// TwinCAT 3 PLC project Plc
// ProgramVersion: 3.1.4023.0
// libraries:
//   Tc2_Standard, * (Beckhoff Automation GmbH)
//   Tc2_System, * (Beckhoff Automation GmbH)
//   Tc3_Module, * (Beckhoff Automation GmbH)
// project tree:
//   / PlcTask.TcTTO (not stored)
//   DUTs/IO/PdoEntries/ Status_3D84275F.TcDUT, Ctrl_1EFB4D3B.TcDUT
//   DUTs/IO/PDOs/ InfoData_6F19DB2B.TcDUT (not stored), COM_TxPDO_Map_Inputs_Channel_3801C95E.TcDUT, COM_TxPDO_Map_Inputs_Channel_6C2FC202.TcDUT, COM_RxPDO_Map_Outputs_Channel_EADA2E0D.TcDUT, COM_RxPDO_Map_Outputs_Channel_5D00B5E7.TcDUT, WcState_9091E0EB.TcDUT, InfoData_32EB74EA.TcDUT, InfoData_E68C61CD.TcDUT (not stored), WcState_0B2B16F9.TcDUT (not stored), InfoData_2A97D6CF.TcDUT (not stored), Inputs_A65FACA4.TcDUT (not stored), Outputs_23C0ED1D.TcDUT (not stored)
//   DUTs/IO/Boxes/ EK1100_1FC0878B.TcDUT (not stored), EL6002_642836E0.TcDUT
//   DUTs/IO/Devices/ SyncUnitTask_2D604ED5.TcDUT (not stored), SyncUnitTasks_6FEB8257.TcDUT (not stored), SyncUnits_99E584AF.TcDUT (not stored)
//   DUTs/IO/Topology/ Term_1_EK1100_40465B6B.TcDUT (not stored), Device_1_EtherCAT_B7DDB641.TcDUT (not stored)
//   DUTs/IO/Base/ EtcSlaveBase_82538BE2.TcDUT (not stored), EtcSlaveBase_82538BE2.TcDUT (not stored), EtcSlaveBase_82538BE2.TcDUT (not stored), EtcSlaveTerminalBase_947E5A46.TcDUT (not stored), EtcSlaveBoxBase_77A0E4A7.TcDUT (not stored), EtcSlaveEndTerminalBase_866C7F0C.TcDUT (not stored), InputBase_8311D824.TcDUT (not stored), OutputBase_10CEE7DE.TcDUT (not stored), EtcMasterBase_62654B43.TcDUT (not stored)
//   GVLs/ GVL_iXlinker.TcGVL (not stored)
// real-time tasks:
//   TASK PlcTask: cycle T#10ms, priority 20, ADS port 350
// I/O:
//   DEVICE Device 1 (EtherCAT), AmsNetId 172.20.30.238.2.1
//     Term 1 (EK1100) [EK1100 EtherCAT Coupler (2A E-Bus)]
//       Term 2 (EL6002) [EL6002 Interface 2Ch. (RS232)]
// variable links:
//   Plc/Plc Instance <-> Device 1 (EtherCAT)/Term 1 (EK1100)
//     PlcTask Inputs/GVL_iXlinker.Device_1_EtherCAT.Term_1_EK1100.InfoData.State <-> InfoData/State
//   Plc/Plc Instance <-> Device 1 (EtherCAT)/Term 1 (EK1100)/Term 2 (EL6002)
//     PlcTask Inputs/GVL_iXlinker.Device_1_EtherCAT.Term_1_EK1100.Term_2_EL6002.COM_TxPDO_Map_Inputs_Channel_1.Status/Transmit_accepted <-> COM TxPDO-Map Inputs Channel 1/Status/Transmit accepted
//     PlcTask Inputs/GVL_iXlinker.Device_1_EtherCAT.Term_1_EK1100.Term_2_EL6002.COM_TxPDO_Map_Inputs_Channel_1.Status/Receive_request <-> COM TxPDO-Map Inputs Channel 1/Status/Receive request
//     PlcTask Inputs/GVL_iXlinker.Device_1_EtherCAT.Term_1_EK1100.Term_2_EL6002.COM_TxPDO_Map_Inputs_Channel_1.Status/Init_accepted <-> COM TxPDO-Map Inputs Channel 1/Status/Init accepted
//     PlcTask Inputs/GVL_iXlinker.Device_1_EtherCAT.Term_1_EK1100.Term_2_EL6002.COM_TxPDO_Map_Inputs_Channel_1.Status/Buffer_full <-> COM TxPDO-Map Inputs Channel 1/Status/Buffer full
//     PlcTask Inputs/GVL_iXlinker.Device_1_EtherCAT.Term_1_EK1100.Term_2_EL6002.COM_TxPDO_Map_Inputs_Channel_1.Status/Parity_error <-> COM TxPDO-Map Inputs Channel 1/Status/Parity error
//     PlcTask Inputs/GVL_iXlinker.Device_1_EtherCAT.Term_1_EK1100.Term_2_EL6002.COM_TxPDO_Map_Inputs_Channel_1.Status/Framing_error <-> COM TxPDO-Map Inputs Channel 1/Status/Framing error
//     PlcTask Inputs/GVL_iXlinker.Device_1_EtherCAT.Term_1_EK1100.Term_2_EL6002.COM_TxPDO_Map_Inputs_Channel_1.Status/Overrun_error <-> COM TxPDO-Map Inputs Channel 1/Status/Overrun error
//     PlcTask Inputs/GVL_iXlinker.Device_1_EtherCAT.Term_1_EK1100.Term_2_EL6002.COM_TxPDO_Map_Inputs_Channel_1.Status/Input_length <-> COM TxPDO-Map Inputs Channel 1/Status/Input length
//     PlcTask Inputs/GVL_iXlinker.Device_1_EtherCAT.Term_1_EK1100.Term_2_EL6002.COM_TxPDO_Map_Inputs_Channel_1.Data_In[0] <-> COM TxPDO-Map Inputs Channel 1/Data In 0
//     PlcTask Inputs/GVL_iXlinker.Device_1_EtherCAT.Term_1_EK1100.Term_2_EL6002.COM_TxPDO_Map_Inputs_Channel_1.Data_In[1] <-> COM TxPDO-Map Inputs Channel 1/Data In 1
//     PlcTask Inputs/GVL_iXlinker.Device_1_EtherCAT.Term_1_EK1100.Term_2_EL6002.COM_TxPDO_Map_Inputs_Channel_1.Data_In[2] <-> COM TxPDO-Map Inputs Channel 1/Data In 2
//     PlcTask Inputs/GVL_iXlinker.Device_1_EtherCAT.Term_1_EK1100.Term_2_EL6002.COM_TxPDO_Map_Inputs_Channel_1.Data_In[3] <-> COM TxPDO-Map Inputs Channel 1/Data In 3
//     PlcTask Inputs/GVL_iXlinker.Device_1_EtherCAT.Term_1_EK1100.Term_2_EL6002.COM_TxPDO_Map_Inputs_Channel_1.Data_In[4] <-> COM TxPDO-Map Inputs Channel 1/Data In 4
//     PlcTask Inputs/GVL_iXlinker.Device_1_EtherCAT.Term_1_EK1100.Term_2_EL6002.COM_TxPDO_Map_Inputs_Channel_1.Data_In[5] <-> COM TxPDO-Map Inputs Channel 1/Data In 5
//     PlcTask Inputs/GVL_iXlinker.Device_1_EtherCAT.Term_1_EK1100.Term_2_EL6002.COM_TxPDO_Map_Inputs_Channel_1.Data_In[6] <-> COM TxPDO-Map Inputs Channel 1/Data In 6
//     PlcTask Inputs/GVL_iXlinker.Device_1_EtherCAT.Term_1_EK1100.Term_2_EL6002.COM_TxPDO_Map_Inputs_Channel_1.Data_In[7] <-> COM TxPDO-Map Inputs Channel 1/Data In 7
//     PlcTask Inputs/GVL_iXlinker.Device_1_EtherCAT.Term_1_EK1100.Term_2_EL6002.COM_TxPDO_Map_Inputs_Channel_1.Data_In[8] <-> COM TxPDO-Map Inputs Channel 1/Data In 8
//     PlcTask Inputs/GVL_iXlinker.Device_1_EtherCAT.Term_1_EK1100.Term_2_EL6002.COM_TxPDO_Map_Inputs_Channel_1.Data_In[9] <-> COM TxPDO-Map Inputs Channel 1/Data In 9
//     PlcTask Inputs/GVL_iXlinker.Device_1_EtherCAT.Term_1_EK1100.Term_2_EL6002.COM_TxPDO_Map_Inputs_Channel_1.Data_In[10] <-> COM TxPDO-Map Inputs Channel 1/Data In 10
//     PlcTask Inputs/GVL_iXlinker.Device_1_EtherCAT.Term_1_EK1100.Term_2_EL6002.COM_TxPDO_Map_Inputs_Channel_1.Data_In[11] <-> COM TxPDO-Map Inputs Channel 1/Data In 11
//     PlcTask Inputs/GVL_iXlinker.Device_1_EtherCAT.Term_1_EK1100.Term_2_EL6002.COM_TxPDO_Map_Inputs_Channel_1.Data_In[12] <-> COM TxPDO-Map Inputs Channel 1/Data In 12
//     PlcTask Inputs/GVL_iXlinker.Device_1_EtherCAT.Term_1_EK1100.Term_2_EL6002.COM_TxPDO_Map_Inputs_Channel_1.Data_In[13] <-> COM TxPDO-Map Inputs Channel 1/Data In 13
//     PlcTask Inputs/GVL_iXlinker.Device_1_EtherCAT.Term_1_EK1100.Term_2_EL6002.COM_TxPDO_Map_Inputs_Channel_1.Data_In[14] <-> COM TxPDO-Map Inputs Channel 1/Data In 14
//     PlcTask Inputs/GVL_iXlinker.Device_1_EtherCAT.Term_1_EK1100.Term_2_EL6002.COM_TxPDO_Map_Inputs_Channel_1.Data_In[15] <-> COM TxPDO-Map Inputs Channel 1/Data In 15
//     PlcTask Inputs/GVL_iXlinker.Device_1_EtherCAT.Term_1_EK1100.Term_2_EL6002.COM_TxPDO_Map_Inputs_Channel_1.Data_In[16] <-> COM TxPDO-Map Inputs Channel 1/Data In 16
//     PlcTask Inputs/GVL_iXlinker.Device_1_EtherCAT.Term_1_EK1100.Term_2_EL6002.COM_TxPDO_Map_Inputs_Channel_1.Data_In[17] <-> COM TxPDO-Map Inputs Channel 1/Data In 17
//     PlcTask Inputs/GVL_iXlinker.Device_1_EtherCAT.Term_1_EK1100.Term_2_EL6002.COM_TxPDO_Map_Inputs_Channel_1.Data_In[18] <-> COM TxPDO-Map Inputs Channel 1/Data In 18
//     PlcTask Inputs/GVL_iXlinker.Device_1_EtherCAT.Term_1_EK1100.Term_2_EL6002.COM_TxPDO_Map_Inputs_Channel_1.Data_In[19] <-> COM TxPDO-Map Inputs Channel 1/Data In 19
//     PlcTask Inputs/GVL_iXlinker.Device_1_EtherCAT.Term_1_EK1100.Term_2_EL6002.COM_TxPDO_Map_Inputs_Channel_1.Data_In[20] <-> COM TxPDO-Map Inputs Channel 1/Data In 20
//     PlcTask Inputs/GVL_iXlinker.Device_1_EtherCAT.Term_1_EK1100.Term_2_EL6002.COM_TxPDO_Map_Inputs_Channel_1.Data_In[21] <-> COM TxPDO-Map Inputs Channel 1/Data In 21
//     PlcTask Inputs/GVL_iXlinker.Device_1_EtherCAT.Term_1_EK1100.Term_2_EL6002.COM_TxPDO_Map_Inputs_Channel_2.Data_In[0] <-> COM TxPDO-Map Inputs Channel 2/Data In 0
//     PlcTask Inputs/GVL_iXlinker.Device_1_EtherCAT.Term_1_EK1100.Term_2_EL6002.COM_TxPDO_Map_Inputs_Channel_2.Data_In[1] <-> COM TxPDO-Map Inputs Channel 2/Data In 1
//     PlcTask Inputs/GVL_iXlinker.Device_1_EtherCAT.Term_1_EK1100.Term_2_EL6002.COM_TxPDO_Map_Inputs_Channel_2.Data_In[2] <-> COM TxPDO-Map Inputs Channel 2/Data In 2
//     PlcTask Inputs/GVL_iXlinker.Device_1_EtherCAT.Term_1_EK1100.Term_2_EL6002.COM_TxPDO_Map_Inputs_Channel_2.Data_In[3] <-> COM TxPDO-Map Inputs Channel 2/Data In 3
//     PlcTask Inputs/GVL_iXlinker.Device_1_EtherCAT.Term_1_EK1100.Term_2_EL6002.COM_TxPDO_Map_Inputs_Channel_2.Data_In[4] <-> COM TxPDO-Map Inputs Channel 2/Data In 4
//     PlcTask Inputs/GVL_iXlinker.Device_1_EtherCAT.Term_1_EK1100.Term_2_EL6002.COM_TxPDO_Map_Inputs_Channel_2.Data_In[5] <-> COM TxPDO-Map Inputs Channel 2/Data In 5
//     PlcTask Inputs/GVL_iXlinker.Device_1_EtherCAT.Term_1_EK1100.Term_2_EL6002.COM_TxPDO_Map_Inputs_Channel_2.Data_In[6] <-> COM TxPDO-Map Inputs Channel 2/Data In 6
//     PlcTask Inputs/GVL_iXlinker.Device_1_EtherCAT.Term_1_EK1100.Term_2_EL6002.COM_TxPDO_Map_Inputs_Channel_2.Data_In[7] <-> COM TxPDO-Map Inputs Channel 2/Data In 7
//     PlcTask Inputs/GVL_iXlinker.Device_1_EtherCAT.Term_1_EK1100.Term_2_EL6002.COM_TxPDO_Map_Inputs_Channel_2.Data_In[8] <-> COM TxPDO-Map Inputs Channel 2/Data In 8
//     PlcTask Inputs/GVL_iXlinker.Device_1_EtherCAT.Term_1_EK1100.Term_2_EL6002.COM_TxPDO_Map_Inputs_Channel_2.Data_In[9] <-> COM TxPDO-Map Inputs Channel 2/Data In 9
//     PlcTask Inputs/GVL_iXlinker.Device_1_EtherCAT.Term_1_EK1100.Term_2_EL6002.COM_TxPDO_Map_Inputs_Channel_2.Data_In[10] <-> COM TxPDO-Map Inputs Channel 2/Data In 10
//     PlcTask Inputs/GVL_iXlinker.Device_1_EtherCAT.Term_1_EK1100.Term_2_EL6002.COM_TxPDO_Map_Inputs_Channel_2.Data_In[11] <-> COM TxPDO-Map Inputs Channel 2/Data In 11
//     PlcTask Inputs/GVL_iXlinker.Device_1_EtherCAT.Term_1_EK1100.Term_2_EL6002.COM_TxPDO_Map_Inputs_Channel_2.Data_In[12] <-> COM TxPDO-Map Inputs Channel 2/Data In 12
//     PlcTask Inputs/GVL_iXlinker.Device_1_EtherCAT.Term_1_EK1100.Term_2_EL6002.COM_TxPDO_Map_Inputs_Channel_2.Data_In[13] <-> COM TxPDO-Map Inputs Channel 2/Data In 13
//     PlcTask Inputs/GVL_iXlinker.Device_1_EtherCAT.Term_1_EK1100.Term_2_EL6002.COM_TxPDO_Map_Inputs_Channel_2.Data_In[14] <-> COM TxPDO-Map Inputs Channel 2/Data In 14
//     PlcTask Inputs/GVL_iXlinker.Device_1_EtherCAT.Term_1_EK1100.Term_2_EL6002.COM_TxPDO_Map_Inputs_Channel_2.Data_In[15] <-> COM TxPDO-Map Inputs Channel 2/Data In 15
//     PlcTask Inputs/GVL_iXlinker.Device_1_EtherCAT.Term_1_EK1100.Term_2_EL6002.COM_TxPDO_Map_Inputs_Channel_2.Data_In[16] <-> COM TxPDO-Map Inputs Channel 2/Data In 16
//     PlcTask Inputs/GVL_iXlinker.Device_1_EtherCAT.Term_1_EK1100.Term_2_EL6002.COM_TxPDO_Map_Inputs_Channel_2.Data_In[17] <-> COM TxPDO-Map Inputs Channel 2/Data In 17
//     PlcTask Inputs/GVL_iXlinker.Device_1_EtherCAT.Term_1_EK1100.Term_2_EL6002.COM_TxPDO_Map_Inputs_Channel_2.Data_In[18] <-> COM TxPDO-Map Inputs Channel 2/Data In 18
//     PlcTask Inputs/GVL_iXlinker.Device_1_EtherCAT.Term_1_EK1100.Term_2_EL6002.COM_TxPDO_Map_Inputs_Channel_2.Data_In[19] <-> COM TxPDO-Map Inputs Channel 2/Data In 19
//     PlcTask Inputs/GVL_iXlinker.Device_1_EtherCAT.Term_1_EK1100.Term_2_EL6002.COM_TxPDO_Map_Inputs_Channel_2.Data_In[20] <-> COM TxPDO-Map Inputs Channel 2/Data In 20
//     PlcTask Inputs/GVL_iXlinker.Device_1_EtherCAT.Term_1_EK1100.Term_2_EL6002.COM_TxPDO_Map_Inputs_Channel_2.Data_In[21] <-> COM TxPDO-Map Inputs Channel 2/Data In 21
//     PlcTask Inputs/GVL_iXlinker.Device_1_EtherCAT.Term_1_EK1100.Term_2_EL6002.COM_TxPDO_Map_Inputs_Channel_2.Status <-> COM TxPDO-Map Inputs Channel 2/Status
//     PlcTask Outputs/GVL_iXlinker.Device_1_EtherCAT.Term_1_EK1100.Term_2_EL6002.COM_RxPDO_Map_Outputs_Channel_1.Ctrl/Transmit_request <-> COM RxPDO-Map Outputs Channel 1/Ctrl/Transmit request
//     PlcTask Outputs/GVL_iXlinker.Device_1_EtherCAT.Term_1_EK1100.Term_2_EL6002.COM_RxPDO_Map_Outputs_Channel_1.Ctrl/Receive_accepted <-> COM RxPDO-Map Outputs Channel 1/Ctrl/Receive accepted
//     PlcTask Outputs/GVL_iXlinker.Device_1_EtherCAT.Term_1_EK1100.Term_2_EL6002.COM_RxPDO_Map_Outputs_Channel_1.Ctrl/Init_request <-> COM RxPDO-Map Outputs Channel 1/Ctrl/Init request
//     PlcTask Outputs/GVL_iXlinker.Device_1_EtherCAT.Term_1_EK1100.Term_2_EL6002.COM_RxPDO_Map_Outputs_Channel_1.Ctrl/Send_continuous <-> COM RxPDO-Map Outputs Channel 1/Ctrl/Send continuous
//     PlcTask Outputs/GVL_iXlinker.Device_1_EtherCAT.Term_1_EK1100.Term_2_EL6002.COM_RxPDO_Map_Outputs_Channel_1.Ctrl/Output_length <-> COM RxPDO-Map Outputs Channel 1/Ctrl/Output length
//     PlcTask Outputs/GVL_iXlinker.Device_1_EtherCAT.Term_1_EK1100.Term_2_EL6002.COM_RxPDO_Map_Outputs_Channel_1.Data_Out[0] <-> COM RxPDO-Map Outputs Channel 1/Data Out 0
//     PlcTask Outputs/GVL_iXlinker.Device_1_EtherCAT.Term_1_EK1100.Term_2_EL6002.COM_RxPDO_Map_Outputs_Channel_1.Data_Out[1] <-> COM RxPDO-Map Outputs Channel 1/Data Out 1
//     PlcTask Outputs/GVL_iXlinker.Device_1_EtherCAT.Term_1_EK1100.Term_2_EL6002.COM_RxPDO_Map_Outputs_Channel_1.Data_Out[2] <-> COM RxPDO-Map Outputs Channel 1/Data Out 2
//     PlcTask Outputs/GVL_iXlinker.Device_1_EtherCAT.Term_1_EK1100.Term_2_EL6002.COM_RxPDO_Map_Outputs_Channel_1.Data_Out[3] <-> COM RxPDO-Map Outputs Channel 1/Data Out 3
//     PlcTask Outputs/GVL_iXlinker.Device_1_EtherCAT.Term_1_EK1100.Term_2_EL6002.COM_RxPDO_Map_Outputs_Channel_1.Data_Out[4] <-> COM RxPDO-Map Outputs Channel 1/Data Out 4
//     PlcTask Outputs/GVL_iXlinker.Device_1_EtherCAT.Term_1_EK1100.Term_2_EL6002.COM_RxPDO_Map_Outputs_Channel_1.Data_Out[5] <-> COM RxPDO-Map Outputs Channel 1/Data Out 5
//     PlcTask Outputs/GVL_iXlinker.Device_1_EtherCAT.Term_1_EK1100.Term_2_EL6002.COM_RxPDO_Map_Outputs_Channel_1.Data_Out[6] <-> COM RxPDO-Map Outputs Channel 1/Data Out 6
//     PlcTask Outputs/GVL_iXlinker.Device_1_EtherCAT.Term_1_EK1100.Term_2_EL6002.COM_RxPDO_Map_Outputs_Channel_1.Data_Out[7] <-> COM RxPDO-Map Outputs Channel 1/Data Out 7
//     PlcTask Outputs/GVL_iXlinker.Device_1_EtherCAT.Term_1_EK1100.Term_2_EL6002.COM_RxPDO_Map_Outputs_Channel_1.Data_Out[8] <-> COM RxPDO-Map Outputs Channel 1/Data Out 8
//     PlcTask Outputs/GVL_iXlinker.Device_1_EtherCAT.Term_1_EK1100.Term_2_EL6002.COM_RxPDO_Map_Outputs_Channel_1.Data_Out[9] <-> COM RxPDO-Map Outputs Channel 1/Data Out 9
//     PlcTask Outputs/GVL_iXlinker.Device_1_EtherCAT.Term_1_EK1100.Term_2_EL6002.COM_RxPDO_Map_Outputs_Channel_1.Data_Out[10] <-> COM RxPDO-Map Outputs Channel 1/Data Out 10
//     PlcTask Outputs/GVL_iXlinker.Device_1_EtherCAT.Term_1_EK1100.Term_2_EL6002.COM_RxPDO_Map_Outputs_Channel_1.Data_Out[11] <-> COM RxPDO-Map Outputs Channel 1/Data Out 11
//     PlcTask Outputs/GVL_iXlinker.Device_1_EtherCAT.Term_1_EK1100.Term_2_EL6002.COM_RxPDO_Map_Outputs_Channel_1.Data_Out[12] <-> COM RxPDO-Map Outputs Channel 1/Data Out 12
//     PlcTask Outputs/GVL_iXlinker.Device_1_EtherCAT.Term_1_EK1100.Term_2_EL6002.COM_RxPDO_Map_Outputs_Channel_1.Data_Out[13] <-> COM RxPDO-Map Outputs Channel 1/Data Out 13
//     PlcTask Outputs/GVL_iXlinker.Device_1_EtherCAT.Term_1_EK1100.Term_2_EL6002.COM_RxPDO_Map_Outputs_Channel_1.Data_Out[14] <-> COM RxPDO-Map Outputs Channel 1/Data Out 14
//     PlcTask Outputs/GVL_iXlinker.Device_1_EtherCAT.Term_1_EK1100.Term_2_EL6002.COM_RxPDO_Map_Outputs_Channel_1.Data_Out[15] <-> COM RxPDO-Map Outputs Channel 1/Data Out 15
//     PlcTask Outputs/GVL_iXlinker.Device_1_EtherCAT.Term_1_EK1100.Term_2_EL6002.COM_RxPDO_Map_Outputs_Channel_1.Data_Out[16] <-> COM RxPDO-Map Outputs Channel 1/Data Out 16
//     PlcTask Outputs/GVL_iXlinker.Device_1_EtherCAT.Term_1_EK1100.Term_2_EL6002.COM_RxPDO_Map_Outputs_Channel_1.Data_Out[17] <-> COM RxPDO-Map Outputs Channel 1/Data Out 17
//     PlcTask Outputs/GVL_iXlinker.Device_1_EtherCAT.Term_1_EK1100.Term_2_EL6002.COM_RxPDO_Map_Outputs_Channel_1.Data_Out[18] <-> COM RxPDO-Map Outputs Channel 1/Data Out 18
//     PlcTask Outputs/GVL_iXlinker.Device_1_EtherCAT.Term_1_EK1100.Term_2_EL6002.COM_RxPDO_Map_Outputs_Channel_1.Data_Out[19] <-> COM RxPDO-Map Outputs Channel 1/Data Out 19
//     PlcTask Outputs/GVL_iXlinker.Device_1_EtherCAT.Term_1_EK1100.Term_2_EL6002.COM_RxPDO_Map_Outputs_Channel_1.Data_Out[20] <-> COM RxPDO-Map Outputs Channel 1/Data Out 20
//     PlcTask Outputs/GVL_iXlinker.Device_1_EtherCAT.Term_1_EK1100.Term_2_EL6002.COM_RxPDO_Map_Outputs_Channel_1.Data_Out[21] <-> COM RxPDO-Map Outputs Channel 1/Data Out 21
//     PlcTask Outputs/GVL_iXlinker.Device_1_EtherCAT.Term_1_EK1100.Term_2_EL6002.COM_RxPDO_Map_Outputs_Channel_2.Data_Out[0] <-> COM RxPDO-Map Outputs Channel 2/Data Out 0
//     PlcTask Outputs/GVL_iXlinker.Device_1_EtherCAT.Term_1_EK1100.Term_2_EL6002.COM_RxPDO_Map_Outputs_Channel_2.Data_Out[1] <-> COM RxPDO-Map Outputs Channel 2/Data Out 1
//     PlcTask Outputs/GVL_iXlinker.Device_1_EtherCAT.Term_1_EK1100.Term_2_EL6002.COM_RxPDO_Map_Outputs_Channel_2.Data_Out[2] <-> COM RxPDO-Map Outputs Channel 2/Data Out 2
//     PlcTask Outputs/GVL_iXlinker.Device_1_EtherCAT.Term_1_EK1100.Term_2_EL6002.COM_RxPDO_Map_Outputs_Channel_2.Data_Out[3] <-> COM RxPDO-Map Outputs Channel 2/Data Out 3
//     PlcTask Outputs/GVL_iXlinker.Device_1_EtherCAT.Term_1_EK1100.Term_2_EL6002.COM_RxPDO_Map_Outputs_Channel_2.Data_Out[4] <-> COM RxPDO-Map Outputs Channel 2/Data Out 4
//     PlcTask Outputs/GVL_iXlinker.Device_1_EtherCAT.Term_1_EK1100.Term_2_EL6002.COM_RxPDO_Map_Outputs_Channel_2.Data_Out[5] <-> COM RxPDO-Map Outputs Channel 2/Data Out 5
//     PlcTask Outputs/GVL_iXlinker.Device_1_EtherCAT.Term_1_EK1100.Term_2_EL6002.COM_RxPDO_Map_Outputs_Channel_2.Data_Out[6] <-> COM RxPDO-Map Outputs Channel 2/Data Out 6
//     PlcTask Outputs/GVL_iXlinker.Device_1_EtherCAT.Term_1_EK1100.Term_2_EL6002.COM_RxPDO_Map_Outputs_Channel_2.Data_Out[7] <-> COM RxPDO-Map Outputs Channel 2/Data Out 7
//     PlcTask Outputs/GVL_iXlinker.Device_1_EtherCAT.Term_1_EK1100.Term_2_EL6002.COM_RxPDO_Map_Outputs_Channel_2.Data_Out[8] <-> COM RxPDO-Map Outputs Channel 2/Data Out 8
//     PlcTask Outputs/GVL_iXlinker.Device_1_EtherCAT.Term_1_EK1100.Term_2_EL6002.COM_RxPDO_Map_Outputs_Channel_2.Data_Out[9] <-> COM RxPDO-Map Outputs Channel 2/Data Out 9
//     PlcTask Outputs/GVL_iXlinker.Device_1_EtherCAT.Term_1_EK1100.Term_2_EL6002.COM_RxPDO_Map_Outputs_Channel_2.Data_Out[10] <-> COM RxPDO-Map Outputs Channel 2/Data Out 10
//     PlcTask Outputs/GVL_iXlinker.Device_1_EtherCAT.Term_1_EK1100.Term_2_EL6002.COM_RxPDO_Map_Outputs_Channel_2.Data_Out[11] <-> COM RxPDO-Map Outputs Channel 2/Data Out 11
//     PlcTask Outputs/GVL_iXlinker.Device_1_EtherCAT.Term_1_EK1100.Term_2_EL6002.COM_RxPDO_Map_Outputs_Channel_2.Data_Out[12] <-> COM RxPDO-Map Outputs Channel 2/Data Out 12
//     PlcTask Outputs/GVL_iXlinker.Device_1_EtherCAT.Term_1_EK1100.Term_2_EL6002.COM_RxPDO_Map_Outputs_Channel_2.Data_Out[13] <-> COM RxPDO-Map Outputs Channel 2/Data Out 13
//     PlcTask Outputs/GVL_iXlinker.Device_1_EtherCAT.Term_1_EK1100.Term_2_EL6002.COM_RxPDO_Map_Outputs_Channel_2.Data_Out[14] <-> COM RxPDO-Map Outputs Channel 2/Data Out 14
//     PlcTask Outputs/GVL_iXlinker.Device_1_EtherCAT.Term_1_EK1100.Term_2_EL6002.COM_RxPDO_Map_Outputs_Channel_2.Data_Out[15] <-> COM RxPDO-Map Outputs Channel 2/Data Out 15
//     PlcTask Outputs/GVL_iXlinker.Device_1_EtherCAT.Term_1_EK1100.Term_2_EL6002.COM_RxPDO_Map_Outputs_Channel_2.Data_Out[16] <-> COM RxPDO-Map Outputs Channel 2/Data Out 16
//     PlcTask Outputs/GVL_iXlinker.Device_1_EtherCAT.Term_1_EK1100.Term_2_EL6002.COM_RxPDO_Map_Outputs_Channel_2.Data_Out[17] <-> COM RxPDO-Map Outputs Channel 2/Data Out 17
//     PlcTask Outputs/GVL_iXlinker.Device_1_EtherCAT.Term_1_EK1100.Term_2_EL6002.COM_RxPDO_Map_Outputs_Channel_2.Data_Out[18] <-> COM RxPDO-Map Outputs Channel 2/Data Out 18
//     PlcTask Outputs/GVL_iXlinker.Device_1_EtherCAT.Term_1_EK1100.Term_2_EL6002.COM_RxPDO_Map_Outputs_Channel_2.Data_Out[19] <-> COM RxPDO-Map Outputs Channel 2/Data Out 19
//     PlcTask Outputs/GVL_iXlinker.Device_1_EtherCAT.Term_1_EK1100.Term_2_EL6002.COM_RxPDO_Map_Outputs_Channel_2.Data_Out[20] <-> COM RxPDO-Map Outputs Channel 2/Data Out 20
//     PlcTask Outputs/GVL_iXlinker.Device_1_EtherCAT.Term_1_EK1100.Term_2_EL6002.COM_RxPDO_Map_Outputs_Channel_2.Data_Out[21] <-> COM RxPDO-Map Outputs Channel 2/Data Out 21
//     PlcTask Outputs/GVL_iXlinker.Device_1_EtherCAT.Term_1_EK1100.Term_2_EL6002.COM_RxPDO_Map_Outputs_Channel_2.Ctrl <-> COM RxPDO-Map Outputs Channel 2/Ctrl
//     PlcTask Inputs/GVL_iXlinker.Device_1_EtherCAT.Term_1_EK1100.Term_2_EL6002.WcState.WcState <-> WcState/WcState
//     PlcTask Inputs/GVL_iXlinker.Device_1_EtherCAT.Term_1_EK1100.Term_2_EL6002.WcState.InputToggle <-> WcState/InputToggle
//     PlcTask Inputs/GVL_iXlinker.Device_1_EtherCAT.Term_1_EK1100.Term_2_EL6002.InfoData.AdsAddr <-> InfoData/AdsAddr
//     PlcTask Inputs/GVL_iXlinker.Device_1_EtherCAT.Term_1_EK1100.Term_2_EL6002.InfoData.State <-> InfoData/State
//   Plc/Plc Instance <-> Device 1 (EtherCAT)
//     PlcTask Inputs/GVL_iXlinker.Device_1_EtherCAT.SyncUnits._default._unreferenced.WcState.WcState <-> SyncUnits/<default>/<unreferenced>/WcState/WcState
//     PlcTask Inputs/GVL_iXlinker.Device_1_EtherCAT.SyncUnits._default._unreferenced.InfoData.ObjectId <-> SyncUnits/<default>/<unreferenced>/InfoData/ObjectId
//     PlcTask Inputs/GVL_iXlinker.Device_1_EtherCAT.SyncUnits._default._unreferenced.InfoData.State <-> SyncUnits/<default>/<unreferenced>/InfoData/State
//     PlcTask Inputs/GVL_iXlinker.Device_1_EtherCAT.SyncUnits._default._unreferenced.InfoData.SlaveCount <-> SyncUnits/<default>/<unreferenced>/InfoData/SlaveCount
//     PlcTask Inputs/GVL_iXlinker.Device_1_EtherCAT.SyncUnits._default.PlcTask.WcState.WcState <-> SyncUnits/<default>/PlcTask/WcState/WcState
//     PlcTask Inputs/GVL_iXlinker.Device_1_EtherCAT.SyncUnits._default.PlcTask.InfoData.ObjectId <-> SyncUnits/<default>/PlcTask/InfoData/ObjectId
//     PlcTask Inputs/GVL_iXlinker.Device_1_EtherCAT.SyncUnits._default.PlcTask.InfoData.State <-> SyncUnits/<default>/PlcTask/InfoData/State
//     PlcTask Inputs/GVL_iXlinker.Device_1_EtherCAT.SyncUnits._default.PlcTask.InfoData.SlaveCount <-> SyncUnits/<default>/PlcTask/InfoData/SlaveCount
//     PlcTask Inputs/GVL_iXlinker.Device_1_EtherCAT.Inputs.SlaveCount <-> Inputs/SlaveCount
//     PlcTask Inputs/GVL_iXlinker.Device_1_EtherCAT.Inputs.DevState <-> Inputs/DevState
//     PlcTask Inputs/GVL_iXlinker.Device_1_EtherCAT.Inputs.Frm0State <-> Inputs/Frm0State
//     PlcTask Inputs/GVL_iXlinker.Device_1_EtherCAT.Inputs.Frm0WcState <-> Inputs/Frm0WcState
//     PlcTask Inputs/GVL_iXlinker.Device_1_EtherCAT.Inputs.Frm0InputToggle <-> Inputs/Frm0InputToggle
//     PlcTask Outputs/GVL_iXlinker.Device_1_EtherCAT.Outputs.DevCtrl <-> Outputs/DevCtrl
//     PlcTask Outputs/GVL_iXlinker.Device_1_EtherCAT.Outputs.Frm0Ctrl <-> Outputs/Frm0Ctrl
//     PlcTask Outputs/GVL_iXlinker.Device_1_EtherCAT.Outputs.Frm0WcCtrl <-> Outputs/Frm0WcCtrl
//     PlcTask Inputs/GVL_iXlinker.Device_1_EtherCAT.InfoData.ChangeCount <-> InfoData/ChangeCount
//     PlcTask Inputs/GVL_iXlinker.Device_1_EtherCAT.InfoData.DevId <-> InfoData/DevId
//     PlcTask Inputs/GVL_iXlinker.Device_1_EtherCAT.InfoData.AmsNetId <-> InfoData/AmsNetId
//     PlcTask Inputs/GVL_iXlinker.Device_1_EtherCAT.InfoData.CfgSlaveCount <-> InfoData/CfgSlaveCount
//     PlcTask Inputs/GVL_iXlinker.Device_1_EtherCAT.InfoData.DcToTcTimeOffset <-> InfoData/DcToTcTimeOffset
//     PlcTask Inputs/GVL_iXlinker.Device_1_EtherCAT.InfoData.DcToExtTimeOffset <-> InfoData/DcToExtTimeOffset

// ---- DUTs/IO/PdoEntries/Status_3D84275F.TcDUT
{attribute 'GeneratedUsingTerminal: EL6002-0000-0019'}
{attribute addProperty BoxType "EL6002-0000-0019"}
{attribute addProperty Id "Transmit_acceptedBOOL1Receive_requestBOOL1Init_acceptedBOOL1Buffer_fullBOOL1Parity_errorBOOL1Framing_errorBOOL1Overrun_errorBOOL1Input_lengthUSINT1"}
{attribute addProperty CRC "1032071007"}
{attribute addProperty Size "8"}
TYPE Status_3D84275F :
STRUCT
	{attribute addProperty Name "Transmit_accepted"}
	Transmit_accepted : BOOL;
	{attribute addProperty Name "Receive_request"}
	Receive_request : BOOL;
	{attribute addProperty Name "Init_accepted"}
	Init_accepted : BOOL;
	{attribute addProperty Name "Buffer_full"}
	Buffer_full : BOOL;
	{attribute addProperty Name "Parity_error"}
	Parity_error : BOOL;
	{attribute addProperty Name "Framing_error"}
	Framing_error : BOOL;
	{attribute addProperty Name "Overrun_error"}
	Overrun_error : BOOL;
	{attribute addProperty Name "Input_length"}
	Input_length : USINT;
END_STRUCT
END_TYPE

// ---- DUTs/IO/PdoEntries/Ctrl_1EFB4D3B.TcDUT
{attribute 'GeneratedUsingTerminal: EL6002-0000-0019'}
{attribute addProperty BoxType "EL6002-0000-0019"}
{attribute addProperty Id "Transmit_requestBOOL1Receive_acceptedBOOL1Init_requestBOOL1Send_continuousBOOL1Output_lengthUSINT1"}
{attribute addProperty CRC "519785787"}
{attribute addProperty Size "5"}
TYPE Ctrl_1EFB4D3B :
STRUCT
	{attribute addProperty Name "Transmit_request"}
	Transmit_request : BOOL;
	{attribute addProperty Name "Receive_accepted"}
	Receive_accepted : BOOL;
	{attribute addProperty Name "Init_request"}
	Init_request : BOOL;
	{attribute addProperty Name "Send_continuous"}
	Send_continuous : BOOL;
	{attribute addProperty Name "Output_length"}
	Output_length : USINT;
END_STRUCT
END_TYPE

// ---- DUTs/IO/PDOs/COM_TxPDO_Map_Inputs_Channel_3801C95E.TcDUT
{attribute 'GeneratedUsingTerminal: EL6002-0000-0019'}
{attribute addProperty BoxType "EL6002-0000-0019"}
{attribute addProperty Id "StatusAT %I*Status_3D84275F8Data_InAT %I*ARRAY[0..21] OF USINT22"}
{attribute addProperty CRC "1334739266"}
{attribute addProperty Size "30"}
TYPE COM_TxPDO_Map_Inputs_Channel_3801C95E EXTENDS InputBase_8311D824 :
STRUCT
	{attribute addProperty Name "Status"}
	Status AT %I* : Status_3D84275F;
	{attribute addProperty Name "Data_In"}
	Data_In AT %I* : ARRAY[0..21] OF USINT;
END_STRUCT
END_TYPE

// ---- DUTs/IO/PDOs/COM_TxPDO_Map_Inputs_Channel_6C2FC202.TcDUT
{attribute 'GeneratedUsingTerminal: EL6002-0000-0019'}
{attribute addProperty BoxType "EL6002-0000-0019"}
{attribute addProperty Id "StatusAT %I*UINT2Data_InAT %I*ARRAY[0..21] OF USINT22"}
{attribute addProperty CRC "1367962124"}
{attribute addProperty Size "24"}
TYPE COM_TxPDO_Map_Inputs_Channel_6C2FC202 EXTENDS InputBase_8311D824 :
STRUCT
	{attribute addProperty Name "Status"}
	Status AT %I* : UINT;
	{attribute addProperty Name "Data_In"}
	Data_In AT %I* : ARRAY[0..21] OF USINT;
END_STRUCT
END_TYPE

// ---- DUTs/IO/PDOs/COM_RxPDO_Map_Outputs_Channel_EADA2E0D.TcDUT
{attribute 'GeneratedUsingTerminal: EL6002-0000-0019'}
{attribute addProperty BoxType "EL6002-0000-0019"}
{attribute addProperty Id "CtrlAT %Q*Ctrl_1EFB4D3B5Data_OutAT %Q*ARRAY[0..21] OF USINT22"}
{attribute addProperty CRC "3494673196"}
{attribute addProperty Size "27"}
TYPE COM_RxPDO_Map_Outputs_Channel_EADA2E0D EXTENDS OutputBase_10CEE7DE :
STRUCT
	{attribute addProperty Name "Ctrl"}
	Ctrl AT %Q* : Ctrl_1EFB4D3B;
	{attribute addProperty Name "Data_Out"}
	Data_Out AT %Q* : ARRAY[0..21] OF USINT;
END_STRUCT
END_TYPE

// ---- DUTs/IO/PDOs/COM_RxPDO_Map_Outputs_Channel_5D00B5E7.TcDUT
{attribute 'GeneratedUsingTerminal: EL6002-0000-0019'}
{attribute addProperty BoxType "EL6002-0000-0019"}
{attribute addProperty Id "CtrlAT %Q*UINT2Data_OutAT %Q*ARRAY[0..21] OF USINT22"}
{attribute addProperty CRC "875731620"}
{attribute addProperty Size "24"}
TYPE COM_RxPDO_Map_Outputs_Channel_5D00B5E7 EXTENDS OutputBase_10CEE7DE :
STRUCT
	{attribute addProperty Name "Ctrl"}
	Ctrl AT %Q* : UINT;
	{attribute addProperty Name "Data_Out"}
	Data_Out AT %Q* : ARRAY[0..21] OF USINT;
END_STRUCT
END_TYPE

// ---- DUTs/IO/PDOs/WcState_9091E0EB.TcDUT
{attribute 'GeneratedUsingTerminal: EL6002-0000-0019'}
{attribute addProperty BoxType "EL6002-0000-0019"}
{attribute addProperty Id "WcStateAT %I*BOOL1InputToggleAT %I*BOOL1"}
{attribute addProperty CRC "2425479403"}
{attribute addProperty Size "2"}
TYPE WcState_9091E0EB :
STRUCT
	{attribute addProperty Name "WcState"}
	WcState AT %I* : BOOL;
	{attribute addProperty Name "InputToggle"}
	InputToggle AT %I* : BOOL;
END_STRUCT
END_TYPE

// ---- DUTs/IO/PDOs/InfoData_32EB74EA.TcDUT
{attribute 'GeneratedUsingTerminal: EL6002-0000-0019'}
{attribute addProperty BoxType "EL6002-0000-0019"}
{attribute addProperty Id "AdsAddrAT %I*AMSADDR8StateAT %I*UINT2"}
{attribute addProperty CRC "854291690"}
{attribute addProperty Size "10"}
TYPE InfoData_32EB74EA EXTENDS InputBase_8311D824 :
STRUCT
	{attribute addProperty Name "AdsAddr"}
	AdsAddr AT %I* : AMSADDR;
	{attribute addProperty Name "State"}
	State AT %I* : UINT;
END_STRUCT
END_TYPE

// ---- DUTs/IO/Boxes/EL6002_642836E0.TcDUT
{attribute 'GeneratedUsingTerminal: EL6002-0000-0019'}
{attribute addProperty BoxType "EL6002-0000-0019"}
{attribute addProperty Description "EL6002 Interface 2Ch. (RS232)"}
{attribute addProperty Physics "KK"}
{attribute addProperty Id "COM_TxPDO_Map_Inputs_Channel_1AT %I*COM_TxPDO_Map_Inputs_Channel_3801C95E30COM_TxPDO_Map_Inputs_Channel_2AT %I*COM_TxPDO_Map_Inputs_Channel_6C2FC20224COM_RxPDO_Map_Outputs_Channel_1AT %Q*COM_RxPDO_Map_Outputs_Channel_EADA2E0D27COM_RxPDO_Map_Outputs_Channel_2AT %Q*COM_RxPDO_Map_Outputs_Channel_5D00B5E724WcStateAT %I*WcState_9091E0EB2InfoDataAT %I*InfoData_32EB74EA10"}
{attribute addProperty CRC "1680357088"}
{attribute addProperty Size "117"}
TYPE EL6002_642836E0 EXTENDS EtcSlaveTerminalBase_947E5A46 :
STRUCT
	{attribute addProperty Name "COM_TxPDO_Map_Inputs_Channel_1"}
	COM_TxPDO_Map_Inputs_Channel_1 : COM_TxPDO_Map_Inputs_Channel_3801C95E;
	{attribute addProperty Name "COM_TxPDO_Map_Inputs_Channel_2"}
	COM_TxPDO_Map_Inputs_Channel_2 : COM_TxPDO_Map_Inputs_Channel_6C2FC202;
	{attribute addProperty Name "COM_RxPDO_Map_Outputs_Channel_1"}
	COM_RxPDO_Map_Outputs_Channel_1 : COM_RxPDO_Map_Outputs_Channel_EADA2E0D;
	{attribute addProperty Name "COM_RxPDO_Map_Outputs_Channel_2"}
	COM_RxPDO_Map_Outputs_Channel_2 : COM_RxPDO_Map_Outputs_Channel_5D00B5E7;
	{attribute addProperty Name "WcState"}
	WcState : WcState_9091E0EB;
	{attribute addProperty Name "InfoData"}
	InfoData : InfoData_32EB74EA;
END_STRUCT
END_TYPE
